// TIA Portal project "proyecto unab" (V16)

(* hardware
DEVICE "S7-1200 station_1"  S7-1200 Station
   slot 0: "Rack_0"  S7-1200 Rack  Rack  V1.0
   slot 1: "PLC_1"  CPU 1211C DC/DC/Rly  6ES7 211-1HE40-0XB0  V4.4
*)

// ===== PLC "PLC_1"  CPU 1211C DC/DC/Rly =====

VAR_GLOBAL   // PLC tag table "Tabla de variables estándar"
   "sañida filtro" AT %MD0 : DWord;
   "Tag_1" AT %M0.0 : Bool;
END_VAR

DATA_BLOCK "Node -Red"   // DB1
{ S7_Optimized_Access := 'FALSE' }
VERSION : 0.1
   VAR
      inicio : Bool;
      parar : Bool;
      "s.planta funcionando" : Bool;
      "valvula emergencia" : Bool;
      "s.bomba agua salada" : Bool;
      "tem,filtro  zeolita" : Time;
      "s,filtro zeolita funcionado" : Bool;
      "s.bomba altapresion" : Bool;
      "barometro presion membranas" : Int;
      "valvula de concentrada hasta optener  800 PSI" : Int;
      "Presión de entrada Aproximada 40 – 50 psi(filtro 5micras)" : DInt;
      "sendor TDS funcionado menor a 250 ppm en 800psi" : DInt;
      "sensor de presion:no más de  900psi y no menor a 15 psi" : Int;
      permeado : Bool;
      cloración : Bool;
      "filtro 5micras" : Bool;
      tds : Bool;
      "and3 salida" : Int;
      "nivel estanque" : DInt;
      "Nivel alto" : Bool;
      "Nivrl Medio" : Bool;
      "Nivel Bajo" : Bool;
      "Alarma Revalse" : Bool;
      "Alarma nivel bajo" : Bool;
      nivel : Int;
      "luz roja nivel alto" : Bool;
      restnivel : Bool;
      modificable : DInt;
      setNivel : Bool;
      "valvula de concentrada hasta optener  800 PSI_1" : DInt;
   END_VAR
BEGIN
END_DATA_BLOCK

// folder: System blocks/Program resources

DATA_BLOCK "tempo,filtro zeolita"   // DB2
{ S7_Optimized_Access := 'TRUE' }
AUTHOR : Simatic
FAMILY : IEC
NAME : IEC_TMR
VERSION : 1.0
// stored: InstanceOfName IEC_TIMER
"IEC_TIMER"
BEGIN
END_DATA_BLOCK

DATA_BLOCK "IEC_Timer_0_DB"   // DB3
{ S7_Optimized_Access := 'TRUE' }
AUTHOR : Simatic
FAMILY : IEC
NAME : IEC_TMR
VERSION : 1.0
// stored: InstanceOfName IEC_TIMER
"IEC_TIMER"
BEGIN
END_DATA_BLOCK

DATA_BLOCK "IEC_Timer_0_DB_1"   // DB4
{ S7_Optimized_Access := 'TRUE' }
AUTHOR : Simatic
FAMILY : IEC
NAME : IEC_TMR
VERSION : 1.0
// stored: InstanceOfName IEC_TIMER
"IEC_TIMER"
BEGIN
END_DATA_BLOCK

DATA_BLOCK "IEC_Timer_0_DB_2"   // DB5
{ S7_Optimized_Access := 'TRUE' }
AUTHOR : Simatic
FAMILY : IEC
NAME : IEC_TMR
VERSION : 1.0
// stored: InstanceOfName IEC_TIMER
"IEC_TIMER"
BEGIN
END_DATA_BLOCK

DATA_BLOCK "IEC_Timer_0_DB_3"   // DB6
{ S7_Optimized_Access := 'TRUE' }
AUTHOR : Simatic
FAMILY : IEC
NAME : IEC_TMR
VERSION : 1.0
// stored: InstanceOfName IEC_TIMER
"IEC_TIMER"
BEGIN
END_DATA_BLOCK

DATA_BLOCK "IEC_Timer_0_DB_4"   // DB8
{ S7_Optimized_Access := 'TRUE' }
AUTHOR : Simatic
FAMILY : IEC
NAME : IEC_TMR
VERSION : 1.0
// stored: InstanceOfName IEC_TIMER
"IEC_TIMER"
BEGIN
END_DATA_BLOCK

DATA_BLOCK "IEC_Timer_0_DB_5"   // DB9
{ S7_Optimized_Access := 'TRUE' }
AUTHOR : Simatic
FAMILY : IEC
NAME : IEC_TMR
VERSION : 1.0
// stored: InstanceOfName IEC_TIMER
"IEC_TIMER"
BEGIN
END_DATA_BLOCK

// folder: (top level)

ORGANIZATION_BLOCK "Main"   // OB1, FBD, ProgramCycle
TITLE = "Main Program Sweep (Cycle)"
{ S7_Optimized_Access := 'TRUE' }
VERSION : 0.1
   VAR_INPUT
      Initial_Call : Bool;   // Initial call of this OB
      Remanence : Bool;   // =True, if remanent data are available
   END_VAR
   VAR_TEMP
      salidat : Time;
      per : Time;
      per2 : Time;
      per4 : Word;
      per5 : Word;
      tem5mi : Int;
      tem5s : DInt;
      s : Time;
   END_VAR
   VAR_TEMP   // added for the SCL form of the ladder/FBD networks
      _w1 : Bool;
   END_VAR
BEGIN

REGION Network 1
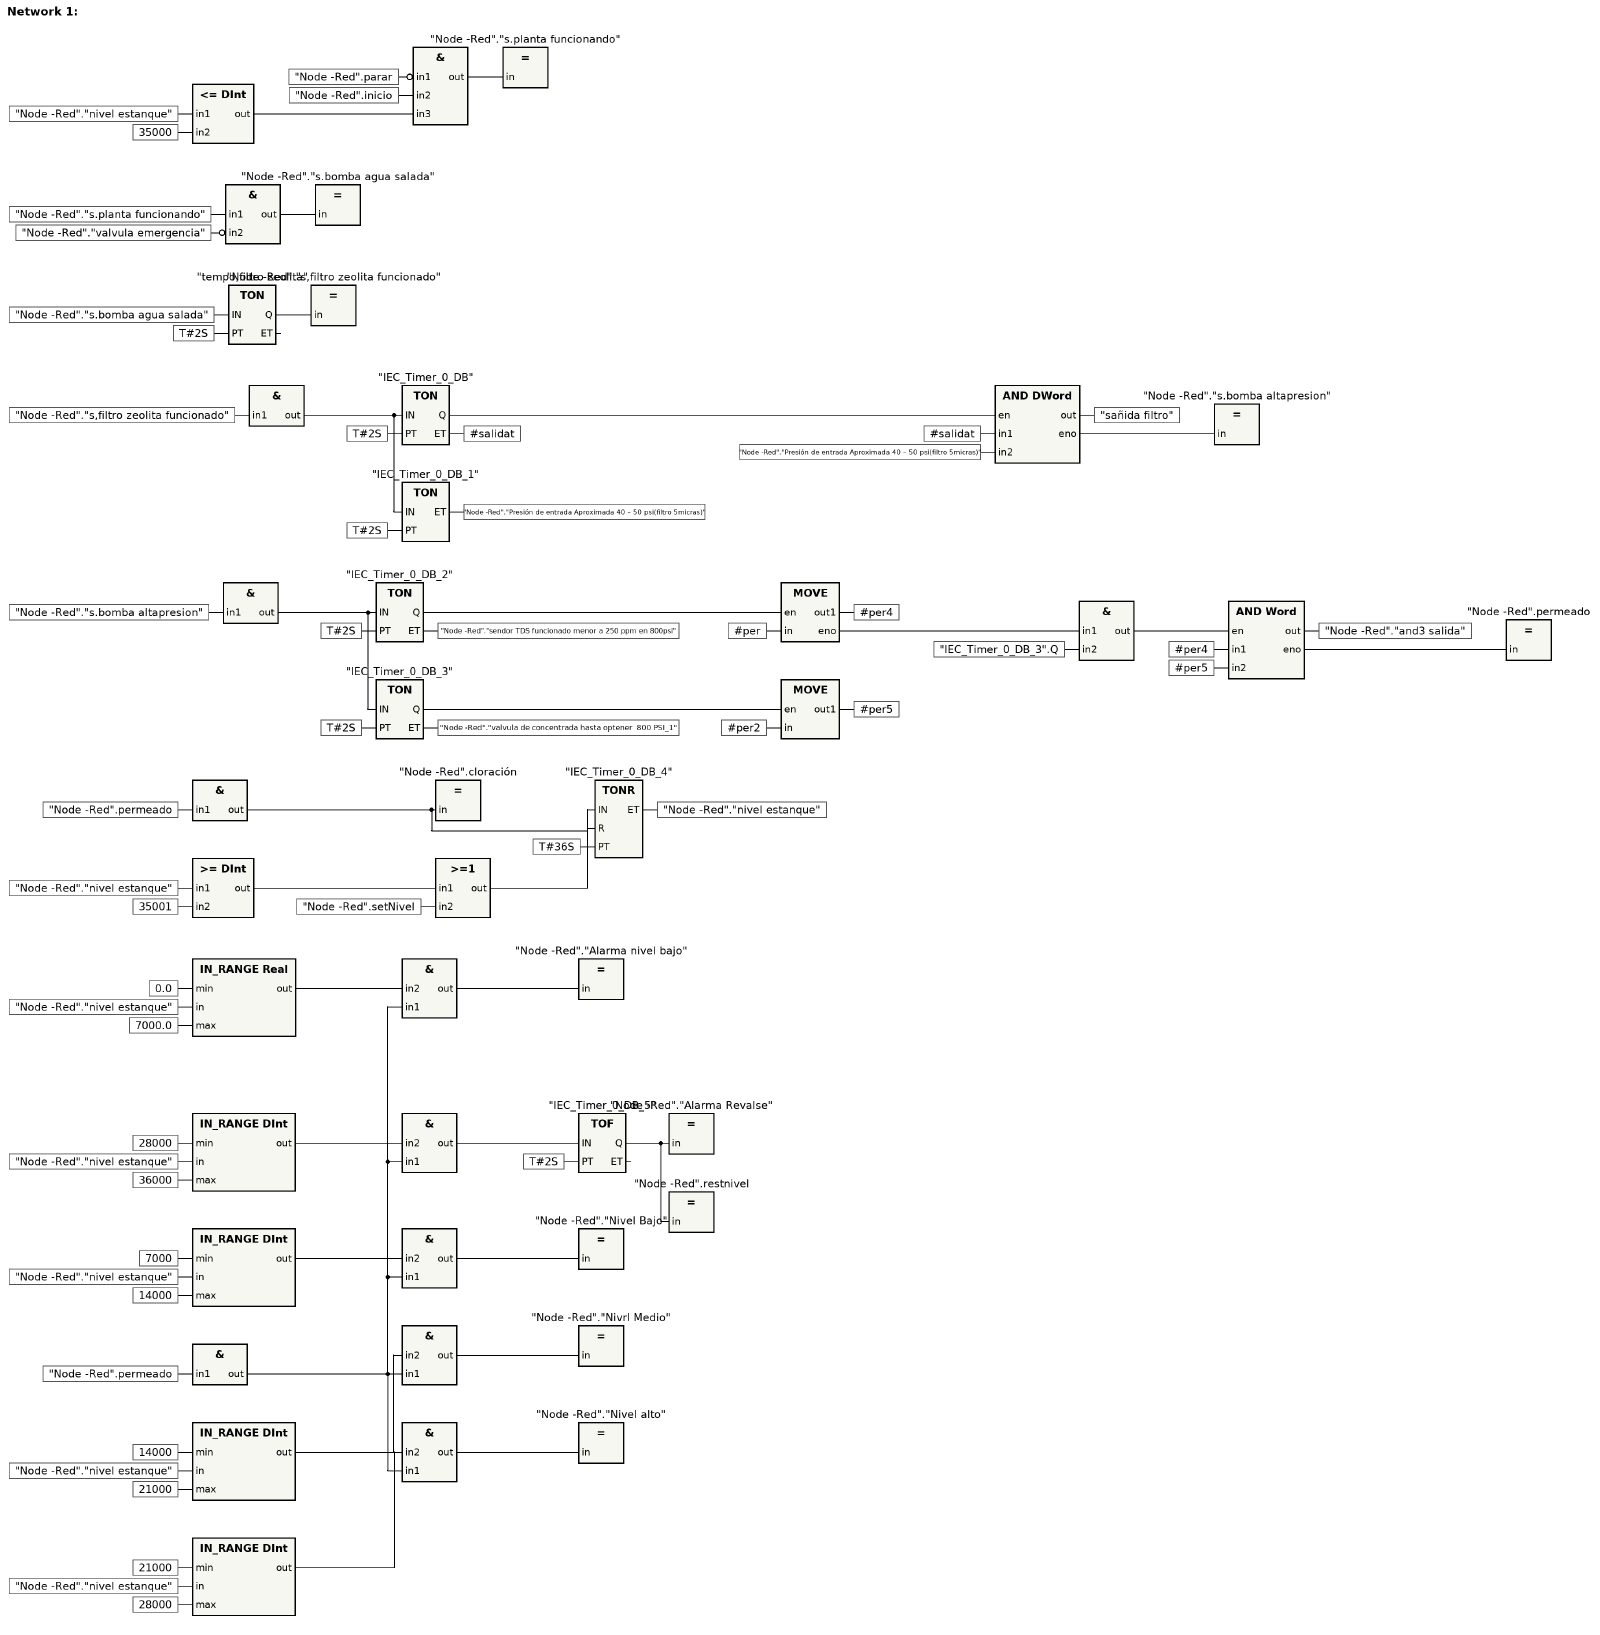
   "Node -Red"."s.planta funcionando" := NOT "Node -Red".parar AND "Node -Red".inicio AND ("Node -Red"."nivel estanque" <= 35000);
   "Node -Red"."s.bomba agua salada" := "Node -Red"."s.planta funcionando" AND NOT "Node -Red"."valvula emergencia";
   "tempo,filtro zeolita".TON(IN := "Node -Red"."s.bomba agua salada", PT := T#2S);
   "Node -Red"."s,filtro zeolita funcionado" := "tempo,filtro zeolita".Q;
   "IEC_Timer_0_DB".TON(IN := "Node -Red"."s,filtro zeolita funcionado", PT := T#2S, ET => #salidat);   // tiempo de espera para encender Bomba de alta
   IF "IEC_Timer_0_DB".Q THEN
       "sañida filtro" := #salidat AND "Node -Red"."Presión de entrada Aproximada 40 – 50 psi(filtro 5micras)";
   END_IF;
   "Node -Red"."s.bomba altapresion" := "IEC_Timer_0_DB".Q;
   "IEC_Timer_0_DB_1".TON(IN := "Node -Red"."s,filtro zeolita funcionado",
                          PT := T#2S,
                          ET => "Node -Red"."Presión de entrada Aproximada 40 – 50 psi(filtro 5micras)");
   "IEC_Timer_0_DB_2".TON(IN := "Node -Red"."s.bomba altapresion",   // sensor TDS funcionado menor a 250 ppm en 800psi
                          PT := T#2S,
                          ET => "Node -Red"."sendor TDS funcionado menor a 250 ppm en 800psi");
   IF "IEC_Timer_0_DB_2".Q THEN #per4 := #per; END_IF;
   #_w1 := "IEC_Timer_0_DB_2".Q AND "IEC_Timer_0_DB_3".Q;
   IF #_w1 THEN "Node -Red"."and3 salida" := #per4 AND #per5; END_IF;
   "Node -Red".permeado := #_w1;
   "IEC_Timer_0_DB_3".TON(IN := "Node -Red"."s.bomba altapresion",   // valvula de concentrada hasta optener 800 PSI
                          PT := T#2S,
                          ET => "Node -Red"."valvula de concentrada hasta optener  800 PSI_1");
   IF "IEC_Timer_0_DB_3".Q THEN #per5 := #per2; END_IF;
   "Node -Red".cloración := "Node -Red".permeado;
   "IEC_Timer_0_DB_4".TONR(IN := "Node -Red".permeado,
                           R := ("Node -Red"."nivel estanque" >= 35001) OR "Node -Red".setNivel,
                           PT := T#36S,
                           ET => "Node -Red"."nivel estanque");
   "Node -Red"."Alarma nivel bajo" := (0.0 <= "Node -Red"."nivel estanque") AND ("Node -Red"."nivel estanque" <= 7000.0) AND "Node -Red".permeado;
   "Node -Red"."Nivel Bajo" := (7000 <= "Node -Red"."nivel estanque") AND ("Node -Red"."nivel estanque" <= 14000) AND "Node -Red".permeado;   // Alarmas
   "Node -Red"."Nivrl Medio" := (14000 <= "Node -Red"."nivel estanque") AND ("Node -Red"."nivel estanque" <= 21000) AND "Node -Red".permeado;
   "Node -Red"."Nivel alto" := (21000 <= "Node -Red"."nivel estanque") AND ("Node -Red"."nivel estanque" <= 28000) AND "Node -Red".permeado;
   "IEC_Timer_0_DB_5".TOF(IN := (28000 <= "Node -Red"."nivel estanque") AND ("Node -Red"."nivel estanque" <= 36000) AND "Node -Red".permeado,
                          PT := T#2S);
   "Node -Red"."Alarma Revalse" := "IEC_Timer_0_DB_5".Q;
   "Node -Red".restnivel := "IEC_Timer_0_DB_5".Q;
END_REGION
END_ORGANIZATION_BLOCK